{attribute 'qualified_only'}
{attribute 'TcHmiSymbol.AddSymbol'}
VAR_GLOBAL PERSISTENT
    // Auto-cycle configuration. PERSISTENT so operator-tuned dwell / timeout
    // values survive an Activate Configuration + PLC restart. Values reset
    // to the struct defaults only on a full cold-boot reset.
    stSepSol1AutoCfg  : ST_HmiPistonAutoCfg;
    stPushSol1AutoCfg : ST_HmiPistonAutoCfg;
END_VAR

(* stored: Version 1.1.0.1, ProductVersion 3.1.4026.18
   GVL GVL_HmiPersistent: Id {b07a24e8-6d3b-41c2-8231-18ba1665c737} *)
